Fanuc KAREL source: pos_grplen.kl

PROGRAM pos_grplen
%NOBUSYLAMP
%NOLOCKGROUP

VAR
	out_reg : INTEGER
%from tpe.klh %import get_int_arg
%from registers.klh %import set_int
%from posetp.klh %import groups_length

BEGIN
	out_reg = tpe__get_int_arg(1)
	registers__set_int(out_reg, posetp__groups_length)
END pos_grplen
